FUNCTION_BLOCK TestStringBufferOutput
VAR_INPUT
END_VAR
VAR_OUTPUT
END_VAR
VAR
  assert: FB_Assert('TestStringBufferOutput');
  
  test_sbo_compose_one_message: StringBufferOutput;
  test_sbo_compose_multiple_messages: StringBufferOutput;
  test_sbo_compose_int_message: StringBufferOutput;
  test_sbo_compose_mixed_messages: StringBufferOutput;
END_VAR

assert.AbortAfterFail := TRUE;
CASE assert.State OF
16#0000:
  IF THIS^.compose_one_message() THEN
    assert.State := assert.State + 16#0010;
	END_IF
16#0010:
  IF THIS^.compose_multiple_messages() THEN
    assert.State := assert.State + 16#0010;
	END_IF
16#0020:
  IF THIS^.compose_int_message() THEN
    assert.State := assert.State + 16#0010;
	END_IF
16#0030:
  IF THIS^.compose_mixed_messages() THEN
    assert.State := assert.State + 16#0010;
	END_IF
16#FFFF:
  ;
ELSE
  assert.PrintPassed('Done');
END_CASE

METHOD compose_int_message : BOOL
VAR_INPUT
END_VAR
VAR
  expected: STRING(10);
  actual: STRING(10);
  
  expected_int: INT;
END_VAR
expected_int := 256;
test_sbo_compose_int_message.compose_message(expected_int);
expected := '256';
actual := test_sbo_compose_int_message.get_output();
compose_int_message := assert.AreEqualSTRING(expected, actual, 'Compose Int message');
END_METHOD

METHOD compose_mixed_messages : BOOL
VAR_INPUT
END_VAR
VAR
  expected: STRING(80);
  actual: STRING(80);
  
  expected_str: STRING(80);
  expected_real: REAL;
  expected_int: INT;
END_VAR
expected_str := 'foo ';
test_sbo_compose_mixed_messages.compose_message(expected_str);
expected_int := -17;
test_sbo_compose_mixed_messages.compose_message(expected_int);
expected_str := ' bar ';
test_sbo_compose_mixed_messages.compose_message(expected_str);
expected_real := 0.1;
test_sbo_compose_mixed_messages.compose_message(expected_real);
expected := 'foo -17 bar 0.1';
actual := test_sbo_compose_mixed_messages.get_output();
compose_mixed_messages := assert.AreEqualSTRING(expected, actual, 'Compose mixed messages');
END_METHOD

METHOD compose_multiple_messages : BOOL
VAR_INPUT
END_VAR
VAR
  expected: STRING(80);
  actual: STRING(80);
  
  expected_str: STRING(80);
END_VAR
expected_str := 'world';
test_sbo_compose_multiple_messages.compose_message(expected_str);
expected_str := 'hello';
test_sbo_compose_multiple_messages.compose_message(expected_str);
expected_str := 'twincat';
test_sbo_compose_multiple_messages.compose_message(expected_str);
expected := 'worldhellotwincat';
actual := test_sbo_compose_multiple_messages.get_output();
compose_multiple_messages := assert.AreEqualSTRING(expected, actual, 'Compose multiple messages');
END_METHOD

METHOD compose_one_message: BOOL
VAR_INPUT
END_VAR
VAR
  expected: STRING(80);
  actual: STRING(80);
  
  expected_str: STRING(80);
END_VAR
expected := 'hello';
test_sbo_compose_one_message.compose_message(expected);
actual := test_sbo_compose_one_message.get_output();
compose_one_message := assert.AreEqualSTRING(expected, actual, 'Compose one message');
END_METHOD

END_FUNCTION_BLOCK

(* stored: Version 1.1.0.1, ProductVersion 3.1.4022.7
   POU TestStringBufferOutput: Id {39f864d9-64bc-4189-b929-64fb5d786ddb}, SpecialFunc None
   Method compose_int_message: Id {41b7c092-1d1b-4aba-888c-715c281ff8cf}
   Method compose_mixed_messages: Id {99792124-7950-46cd-aa60-5b99326f8ee8}
   Method compose_multiple_messages: Id {96f3da7f-eac2-4527-a977-32d5a6dcfba7}
   Method compose_one_message: Id {6bee1a68-a4e2-4600-b4de-d6f5bcbc109c} *)
